{attribute 'qualified_only'}
VAR_GLOBAL
	uReadData_TcpExchangeTask: Int;
	uWriteData_PlcTask: Int;
END_VAR

(* stored: Version 1.1.0.1, ProductVersion 3.1.4024.12
   GVL GVL_TcpExchange: Id {d5718940-a042-46e1-926a-fbeed7b7a419} *)
